// TIA Portal V18 export
FUNCTION_BLOCK "Emergency_Block"   // FB3, SCL
{ S7_Optimized_Access := 'TRUE' }
VERSION : 0.1
// stored: AutoNumber true, IsIECCheckEnabled false, IsRetainMemResEnabled false, MemoryReserve 100, SetENOAutomatically false, UDAEnableTagReadback false
   VAR_OUTPUT
      emergency_state : Bool;
   END_VAR
BEGIN
   REGION Variables OF Emergency timers in Integer (TO show on HMI)
       "Var".Emer_timer_noFlow_int := TIME_TO_INT("Var".Emer_timer_noFlow);
       "Var".Emer_timer_Flow_int := TIME_TO_INT("Var".Emer_timer_Flow);
       "Var".Emer_timer_FCV_closed_int := TIME_TO_INT("Var".Emer_timer_FCV_closed);
       "Var".Emer_timer_ESD_closed_int := TIME_TO_INT("Var".Emer_timer_ESD_closed);
       "Var".Emer_timer_FCV_Open_int := TIME_TO_INT("Var".Emer_timer_FCV_Open);
       "Var".Emer_timer_ESD_Open_int := TIME_TO_INT("Var".Emer_timer_ESD_Open);
   END_REGION

   REGION Assign the emergencies


       // Emergency 1,*******************************************************************************************************
       REGION Emergency 1, fungo
           "Emergency_DB".Emergency_1 := NOT "emergency_mushroom";
       END_REGION

       // Emergency 2,*******************************************************************************************************
       REGION Emergency 2, pendant Emergency
           "Emergency_DB".Emergency_2 := NOT "pendant_emergency_stop";
       END_REGION

       // Emergency 3,*******************************************************************************************************
       REGION Emergency 3, Grounding
           "Emergency_DB".Emergency_3 := (NOT "ground_monitor_IBC") AND ("Var".loading_flag OR "Var".draining_flag);
       END_REGION

       // Emergency 4,*******************************************************************************************************
       REGION Emergency 4, High Level Switch
           "Emergency_DB".Emergency_4 := NOT "Capacitive_HLS";
       END_REGION

       // Emergency 5,*******************************************************************************************************
       REGION Emergency 5, Temperature
           "Emergency_DB".Emergency_5 := ("Temperature_RTD" / 10) > "Var".temperature_threshold AND "Temperature_RTD" < 29000;
       END_REGION

       // Emergency 6,******************************************************************************************************
       REGION Emergency 6, no flow in the loading state 
           IF "Var".loading_flag THEN

               "IEC_Timer_0_DB_5".TON(IN := "flowmeter_analog_feedback" < 1000,
                                      PT := "Var".Emer_timer_noFlow);

               IF "IEC_Timer_0_DB_5".Q THEN
                   "Emergency_DB".Emergency_6 := 1;
               END_IF;

           ELSE
               "Emergency_DB".Emergency_6 := 0;
           END_IF;

           IF NOT "Var".loading_flag OR "flowmeter_analog_feedback" > 1000 THEN
               RESET_TIMER("IEC_Timer_0_DB_5");
           END_IF;

       END_REGION

       // Emergency 7,******************************************************************************************************
       REGION Emergency 7, having flow in no flow state
           IF "Var".no_flow_states THEN

               "IEC_Timer_0_DB_11".TON(IN := "flowmeter_analog_feedback" > 50 AND "flowmeter_analog_feedback" < 29000,
                                       PT := "Var".Emer_timer_Flow);
               //If it is greater than the minimum (there is flow) after 3 seconds of being in Idle
               // the FLOW condition, can be changed!
               IF "IEC_Timer_0_DB_11".Q THEN
                   "Emergency_DB".Emergency_7 := 1;
               END_IF;
           END_IF;

           // reset its related timer 
           IF NOT ("flowmeter_analog_feedback" > 50 AND "flowmeter_analog_feedback" < 29000) OR NOT "Var".no_flow_states THEN

               "Emergency_DB".Emergency_7 := 0;
               RESET_TIMER("IEC_Timer_0_DB_11");
           END_IF;
       END_REGION

       // Emergency 8,*****************************************************************************************************
       REGION Emergency 8, FCV closed in loading
           IF "Var".loading_flag THEN

               //after 7 seconds being in loading and still the FCV is closed. 
               "IEC_Timer_0_DB_10".TON(IN := "FCV_valve_closed",
                                       PT := "Var".Emer_timer_FCV_closed);

               IF "IEC_Timer_0_DB_10".Q THEN
                   "Emergency_DB".Emergency_8 := 1;
               END_IF;
           ELSE
               "Emergency_DB".Emergency_8 := 0;
           END_IF;
           //resets the related timer 
           IF NOT "Var".loading_flag OR "FCV_valve_closed" THEN
               RESET_TIMER("IEC_Timer_0_DB_10");
           END_IF;
       END_REGION

       // Emergency 9,******************************************************************************************************
       REGION Emergency 9, ESD closed in loading
           IF "Var".loading_flag THEN
               //after 3 seconds being in loading and still the ESD is closed. 
               "IEC_Timer_0_DB_13".TON(IN := "ESD_valve_closed",
                                       PT := "Var".Emer_timer_ESD_closed);

               IF "IEC_Timer_0_DB_13".Q THEN

                   "Emergency_DB".Emergency_9 := 1;
               END_IF;
           END_IF;

           // If you are not in loading or ESD valve is not cloesed, this emergency should be reset.
           IF NOT "ESD_valve_closed" OR NOT "Var".loading_flag THEN
               RESET_TIMER("IEC_Timer_0_DB_13");
               "Emergency_DB".Emergency_9 := 0;
           END_IF;

       END_REGION

       //Emergency 10 **************************************************************************************************
       REGION Emergency 10, ESD open in no flow
           "IEC_Timer_0_DB".TON(IN := "Var".no_flow_states AND ("ESD_valve_open" OR NOT "ESD_valve_closed"),
                                PT := "Var".Emer_timer_ESD_Open);

           IF "IEC_Timer_0_DB".Q THEN
               "Emergency_DB".Emergency_10 := 1;
           END_IF;

           // Reseting the ESD valve Open timer
           IF NOT ("Var".no_flow_states AND ("ESD_valve_open" OR NOT "ESD_valve_closed")) THEN

               RESET_TIMER("IEC_Timer_0_DB");
               "Emergency_DB".Emergency_10 := 0;

           END_IF;
       END_REGION

       //Emergency 11 ***************************************************************************************************
       REGION emergency 11, FCV open in no flow

           "IEC_Timer_0_DB_1".TON(IN := "Var".no_flow_states AND ("FCV_valve_open" OR NOT "FCV_valve_closed"),
                                  PT := "Var".Emer_timer_FCV_Open);

           IF "IEC_Timer_0_DB_1".Q THEN
               "Emergency_DB".Emergency_11 := 1;
           END_IF;

           //reseting the FCV valve open timer
           IF NOT ("Var".no_flow_states AND ("FCV_valve_open" OR NOT "FCV_valve_closed")) THEN

               RESET_TIMER("IEC_Timer_0_DB_1");
               "Emergency_DB".Emergency_11 := 0;

           END_IF;
       END_REGION

       //Emergency 12,*****************************************************************************************************
       REGION Emergency 12, the cable OF flowmeter is disconnected


           //Flowmeter after 5 seconds of being disconnected, rises an alarm
           "IEC_Timer_0_DB_8".TON(IN:="flowmeter_analog_feedback" > 30000,
                                  PT:=T#10s);
           IF "IEC_Timer_0_DB_8".Q THEN
               "Emergency_DB".Emergency_12 := 1;
           END_IF;

           IF "flowmeter_analog_feedback" < 30000 THEN
               "Emergency_DB".Emergency_12 := 0;
               RESET_TIMER("IEC_Timer_0_DB_8");

           END_IF;


       END_REGION

       //Emergency 13******************************************************************************************************
       REGION Emergency 13, the cable OF RTD is disconnected

           //RTD after 5 seconds of being disconnected, rises an alarm

           "IEC_Timer_0_DB_7".TON(IN:="Temperature_RTD" > 30000,
                                  PT:=T#5s);
           IF "IEC_Timer_0_DB_7".Q THEN
               "Emergency_DB".Emergency_13 := 1;
           END_IF;


           IF "Temperature_RTD" < 30000 THEN
               "Emergency_DB".Emergency_13 := 0;
               RESET_TIMER("IEC_Timer_0_DB_7");
           END_IF;


       END_REGION

   END_REGION


   REGION Going TO Emergency
       //The #emergencies defined above
       #emergency_state := NOT (
       "Emergency_DB".Emergency_1
       OR "Emergency_DB".Emergency_2
       OR "Emergency_DB".Emergency_3 // Grounding only in flow state should be considered
       OR "Emergency_DB".Emergency_4
       OR "Emergency_DB".Emergency_5
       OR "Emergency_DB".Emergency_6
       OR "Emergency_DB".Emergency_7
       OR "Emergency_DB".Emergency_8
       OR "Emergency_DB".Emergency_9
       OR "Emergency_DB".Emergency_10
       OR "Emergency_DB".Emergency_11
       OR "Emergency_DB".Emergency_12
       OR "Emergency_DB".Emergency_13);

   END_REGION



   //1 FOR NO EMERGENCY, 0 IN CASE OF EMERGENCY
   // These are the flags only for the HMI pop up
   // To prevent from showing multiple emergencies on top, ELSIF is utilized
   REGION Emergency TO HMI
       //when there is an emergency, just set them immediately
       IF #emergency_state = 0 AND "Emergency_DB".Emergency_1 THEN 
           "Emergency_DB".Emergency_1_flag := "Emergency_DB".Emergency_1;

       ELSIF #emergency_state = 0 AND "Emergency_DB".Emergency_2 THEN
           "Emergency_DB".Emergency_2_flag := "Emergency_DB".Emergency_2;

       ELSIF #emergency_state = 0 AND "Emergency_DB".Emergency_3 THEN
           "Emergency_DB".Emergency_3_flag := "Emergency_DB".Emergency_3;

       ELSIF #emergency_state = 0 AND "Emergency_DB".Emergency_4 THEN
           "Emergency_DB".Emergency_4_flag := "Emergency_DB".Emergency_4;

       ELSIF #emergency_state = 0 AND "Emergency_DB".Emergency_5 THEN  
           "Emergency_DB".Emergency_5_flag := "Emergency_DB".Emergency_5;

       ELSIF #emergency_state = 0 AND "Emergency_DB".Emergency_6 THEN
           "Emergency_DB".Emergency_6_flag := "Emergency_DB".Emergency_6;

       ELSIF #emergency_state = 0 AND "Emergency_DB".Emergency_7 THEN
           "Emergency_DB".Emergency_7_flag := "Emergency_DB".Emergency_7;

       ELSIF #emergency_state = 0 AND "Emergency_DB".Emergency_8 THEN
           "Emergency_DB".Emergency_8_flag := "Emergency_DB".Emergency_8;

       ELSIF #emergency_state = 0 AND "Emergency_DB".Emergency_9 THEN
           "Emergency_DB".Emergency_9_flag := "Emergency_DB".Emergency_9;

       ELSIF #emergency_state = 0 AND "Emergency_DB".Emergency_10 THEN
           "Emergency_DB".Emergency_10_flag := "Emergency_DB".Emergency_10;

       ELSIF #emergency_state = 0 AND "Emergency_DB".Emergency_11 THEN
           "Emergency_DB".Emergency_11_flag := "Emergency_DB".Emergency_11;

       ELSIF #emergency_state = 0 AND "Emergency_DB".Emergency_12 THEN
           "Emergency_DB".Emergency_12_flag := "Emergency_DB".Emergency_12;

       ELSIF #emergency_state = 0 AND "Emergency_DB".Emergency_13 THEN
           "Emergency_DB".Emergency_13_flag := "Emergency_DB".Emergency_13;
       END_IF;

       // if the emergency is solved, then by pressing enter ,reset them
       IF "ENTER_Button" THEN
           "Emergency_DB".Emergency_1_flag  := "Emergency_DB".Emergency_1;
           "Emergency_DB".Emergency_2_flag  := "Emergency_DB".Emergency_2;
           "Emergency_DB".Emergency_3_flag  := "Emergency_DB".Emergency_3;
           "Emergency_DB".Emergency_4_flag  := "Emergency_DB".Emergency_4;
           "Emergency_DB".Emergency_5_flag  := "Emergency_DB".Emergency_5;
           "Emergency_DB".Emergency_6_flag  := "Emergency_DB".Emergency_6;
           "Emergency_DB".Emergency_7_flag  := "Emergency_DB".Emergency_7;
           "Emergency_DB".Emergency_8_flag  := "Emergency_DB".Emergency_8;
           "Emergency_DB".Emergency_9_flag  := "Emergency_DB".Emergency_9;
           "Emergency_DB".Emergency_10_flag := "Emergency_DB".Emergency_10;
           "Emergency_DB".Emergency_11_flag := "Emergency_DB".Emergency_11; 
           "Emergency_DB".Emergency_12_flag := "Emergency_DB".Emergency_12;
           "Emergency_DB".Emergency_13_flag := "Emergency_DB".Emergency_13;
           ;
       END_IF;
   END_REGION
END_FUNCTION_BLOCK
